Yaskawa INFORM job: t_01_08_23_cylinder_program.JBI

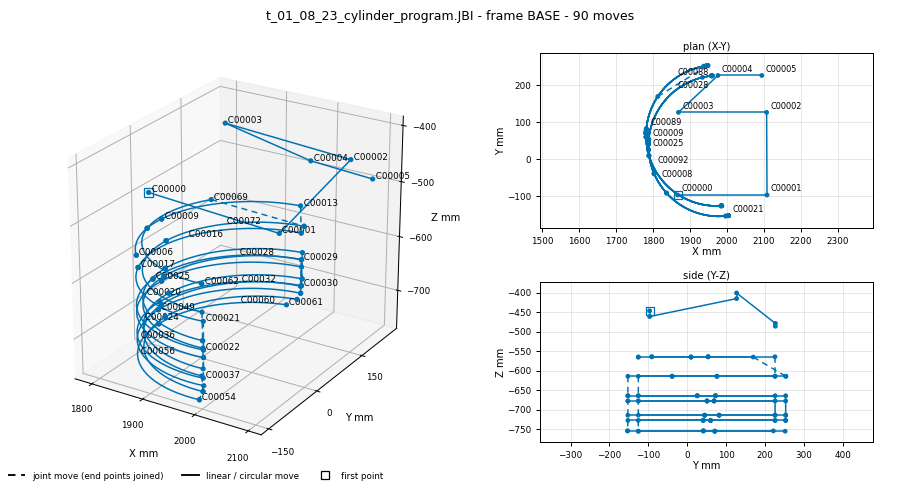
[picture p0: tool path of t_01_08_23_cylinder_program.JBI in frame BASE, 90 of 125 moves have a stored position in this frame; points joined in program order, loops and branches not executed]
/JOB
//NAME t_01_08_23_cylinder_program
//POS
///NPOS 118,0,118,0,0,0
///TOOL 0
///POSTYPE BASE
///RECTAN
///RCONF 0,0,0,0,0,0,0,0,0,0,0,0,0,0,0,0,0,0,0,0,0,0,0,0
C00000=1866.907856,-96.774129,-446.002528,175.000000,-50.248348,92.918411
C00001=2108.409771,-96.774089,-460.785696,175.000000,-50.248348,92.918411
C00002=2107.340894,126.546568,-414.757146,152.980956,5.000000,-5.000000
C00003=1869.210666,126.546528,-400.180371,152.980956,5.000000,-5.000000
C00004=1975.714402,226.206036,-478.423517,175.000000,-60.000000,-90.532197
C00005=2094.376869,226.206056,-485.687257,175.000000,-60.000000,-90.532197
C00006=1836.815666,-91.346481,-564.151000,-138.035050,-90.000000,5.000000
C00007=1836.815666,-91.346481,-564.151000,-138.035050,-90.000000,5.000000
C00008=1813.462641,-59.170193,-564.151000,-150.021884,-90.000000,5.000000
C00009=1788.802698,53.507037,-564.151000,174.711510,-90.000000,5.000000
C00010=1788.802698,53.507037,-564.151000,174.711510,-90.000000,5.000000
C00011=1788.802698,53.507037,-564.151000,174.711510,-90.000000,5.000000
C00012=1799.194788,100.302609,-564.151000,160.247038,-89.999999,5.000000
C00013=1957.618472,225.208793,-564.151000,96.259663,-90.000000,5.000000
C00014=1959.368351,225.392556,-614.195000,95.730143,-89.999999,5.000000
C00015=1959.368351,225.392556,-614.195000,95.730143,-89.999999,5.000000
C00016=1801.888713,107.361045,-614.195000,157.973217,-90.000000,5.000000
C00017=1803.351040,-38.955819,-614.195000,-156.827998,-90.000000,5.000000
C00018=1803.351040,-38.955819,-614.195000,-156.827998,-90.000000,5.000000
C00019=1803.351040,-38.955819,-614.195000,-156.827998,-90.000000,5.000000
C00020=1871.671478,-121.712228,-614.195000,-124.088520,-90.000000,5.000000
C00021=2004.609733,-152.609584,-614.195000,-82.080123,-89.999999,5.000000
C00022=2004.545282,-152.618539,-664.237500,-82.099706,-89.999999,5.000000
C00023=2004.545282,-152.618539,-664.237500,-82.099706,-89.999999,5.000000
C00024=1861.423248,-114.267854,-664.237500,-127.901229,-90.000000,5.000000
C00025=1788.282629,25.448540,-664.237500,-175.000000,-90.000000,5.000000
C00026=1788.282629,25.448540,-664.237500,-175.000000,-90.000000,5.000000
C00027=1788.282629,25.448540,-664.237500,-175.000000,-90.000000,5.000000
C00028=1857.406269,182.970813,-664.237500,129.449763,-90.000000,5.000000
C00029=1960.228639,225.476909,-664.237500,95.470000,-89.999999,5.000000
C00030=1959.424752,225.398207,-714.244000,95.713085,-90.000000,5.000000
C00031=1959.424752,225.398207,-714.244000,95.713085,-90.000000,5.000000
C00032=1860.043911,185.102125,-714.244000,128.429203,-90.000000,5.000000
C00033=1788.186763,44.562490,-714.244000,175.000000,-89.999999,5.000000
C00034=1788.186763,44.562490,-714.244000,175.000000,-89.999999,5.000000
C00035=1788.186763,44.562490,-714.244000,175.000000,-89.999999,5.000000
C00036=1834.273085,-88.461094,-714.244000,-139.192453,-90.000000,5.000000
C00037=2003.923519,-152.703775,-714.244000,-82.288574,-90.000000,5.000000
C00038=2004.586601,-152.612801,-677.657460,-175.000000,-60.000000,97.912848
C00039=2004.586601,-152.612801,-677.657460,-175.000000,-60.000000,97.912848
C00040=1828.234217,-81.102716,-677.657460,175.000000,-60.000000,37.942494
C00041=1788.560641,50.659282,-677.657460,175.000000,-60.000000,-5.000000
C00042=1788.560641,50.659282,-677.657460,175.000000,-60.000000,-5.000000
C00043=1788.560641,50.659282,-677.657460,175.000000,-60.000000,-5.000000
C00044=1853.077163,179.298948,-677.657460,-175.000000,-60.000000,-48.841817
C00045=1960.796933,225.530469,-677.657460,175.000000,-60.000000,-84.701785
C00046=1959.683285,225.423893,-727.621460,175.000000,-60.000000,-84.365103
C00047=1959.683285,225.423893,-727.621460,175.000000,-60.000000,-84.365103
C00048=1855.996123,181.799021,-727.621460,175.000000,-60.000000,-49.998458
C00049=1788.052126,40.732629,-727.621460,-175.000000,-60.000000,-5.000000
C00050=1788.052126,40.732629,-727.621460,-175.000000,-60.000000,-5.000000
C00051=1788.052126,40.732629,-727.621460,-175.000000,-60.000000,-5.000000
C00052=1823.090180,-74.187752,-727.621460,175.000000,-60.000000,35.348569
C00053=2004.520010,-152.622044,-727.621460,175.000000,-60.000000,97.892616
C00054=1996.799177,-153.532136,-754.534960,175.000000,-60.000000,95.552802
C00055=1996.799177,-153.532136,-754.534960,175.000000,-60.000000,95.552802
C00056=1821.172558,-71.433123,-754.534960,175.000000,-60.000000,34.338464
C00057=1788.066435,41.272587,-754.534960,175.000000,-60.000000,-5.000000
C00058=1788.066435,41.272587,-754.534960,175.000000,-60.000000,-5.000000
C00059=1788.066435,41.272587,-754.534960,175.000000,-60.000000,-5.000000
C00060=1858.465261,183.835862,-754.534960,175.000000,-60.000000,-50.961753
C00061=1934.046589,221.110871,-754.534960,175.000000,-60.000000,-76.535293
C00062=1984.729913,-125.856900,-564.850500,-86.117270,-90.000000,5.000000
C00063=1984.729913,-125.856900,-564.850500,-86.117270,-90.000000,5.000000
C00064=1823.365128,-55.081799,-564.850500,-141.247545,-90.000000,5.000000
C00065=1789.445749,9.507244,-564.850500,-163.339420,-90.000000,5.000000
C00066=1789.445749,9.507244,-564.850500,-163.339420,-90.000000,5.000000
C00067=1789.445749,9.507244,-564.850500,-163.339420,-90.000000,5.000000
C00068=1781.565163,70.613527,-564.850500,175.000000,-90.000000,5.000000
C00069=1813.170254,169.308927,-564.850500,146.450271,-90.000000,5.000000
C00070=1948.855670,253.083256,-614.253000,96.933410,-90.000000,5.000000
C00071=1948.855670,253.083256,-614.253000,96.933410,-90.000000,5.000000
C00072=1827.501897,188.241517,-614.253000,139.299547,-89.999999,5.000000
C00073=1781.843312,76.269362,-614.253000,175.000000,-90.000000,5.000000
C00074=1781.843312,76.269362,-614.253000,175.000000,-90.000000,5.000000
C00075=1781.843312,76.269362,-614.253000,175.000000,-90.000000,5.000000
C00076=1839.012225,-72.304280,-614.253000,-134.240439,-89.999999,5.000000
C00077=1984.854502,-125.848403,-614.253000,-86.079688,-89.999999,5.000000
C00078=1985.670166,-125.790746,-664.261500,-85.833603,-90.000000,5.000000
C00079=1985.670166,-125.790746,-664.261500,-85.833603,-90.000000,5.000000
C00080=1817.484848,-47.360560,-664.261500,-144.168682,-89.999999,5.000000
C00081=1781.629678,72.281824,-664.261500,175.000000,-90.000000,5.000000
C00082=1781.629678,72.281824,-664.261500,175.000000,-90.000000,5.000000
C00083=1781.629678,72.281824,-664.261500,175.000000,-90.000000,5.000000
C00084=1848.588115,209.196904,-664.261500,130.343854,-90.000000,5.000000
C00085=1946.287238,252.753181,-664.261500,97.712735,-90.000000,5.000000
C00086=1946.337263,252.759949,-714.232500,97.697544,-89.999999,5.000000
C00087=1946.337263,252.759949,-714.232500,97.697544,-89.999999,5.000000
C00088=1857.182730,216.079242,-714.232500,127.029772,-90.000000,5.000000
C00089=1782.269209,81.696835,-714.232500,174.693933,-89.999999,5.000000
C00090=1782.269209,81.696835,-714.232500,174.693933,-89.999999,5.000000
C00091=1782.269209,81.696835,-714.232500,174.693933,-89.999999,5.000000
C00092=1801.115148,-20.170739,-714.232500,-153.731021,-90.000000,5.000000
C00093=1986.144740,-125.755579,-714.232500,-85.690389,-89.999999,5.000000
C00094=1986.131450,-125.756580,-677.631960,175.000000,-60.000000,94.305599
C00095=1986.131450,-125.756580,-677.631960,175.000000,-60.000000,94.305599
C00096=1813.820766,-42.101735,-677.631960,-175.000000,-60.000000,33.902326
C00097=1781.507638,68.635230,-677.631960,175.000000,-60.000000,-5.000000
C00098=1781.507638,68.635230,-677.631960,175.000000,-60.000000,-5.000000
C00099=1781.507638,68.635230,-677.631960,175.000000,-60.000000,-5.000000
C00100=1843.052224,204.306842,-677.631960,175.000000,-60.000000,-47.433091
C00101=1945.255131,252.610524,-677.631960,175.000000,-60.000000,-81.973701
C00102=1945.341344,252.622661,-727.629960,175.000000,-60.000000,-81.999903
C00103=1945.341344,252.622661,-727.629960,175.000000,-60.000000,-81.999903
C00104=1840.373702,201.798651,-727.629960,175.000000,-60.000000,-46.328736
C00105=1781.500906,59.837692,-727.629960,175.000000,-60.000000,5.000000
C00106=1781.500906,59.837692,-727.629960,175.000000,-60.000000,5.000000
C00107=1781.500906,59.837692,-727.629960,175.000000,-60.000000,5.000000
C00108=1812.240335,-39.711348,-727.629960,175.000000,-60.000000,33.039921
C00109=1983.737597,-125.921646,-727.629960,175.000000,-60.000000,93.583460
C00110=1985.619988,-125.794394,-755.330960,175.000000,-60.000000,94.151256
C00111=1985.619988,-125.794394,-755.330960,175.000000,-60.000000,94.151256
C00112=1814.137027,-42.570833,-755.330960,175.000000,-60.000000,34.072588
C00113=1781.563747,70.572080,-755.330960,175.000000,-60.000000,-5.000000
C00114=1781.563747,70.572080,-755.330960,175.000000,-60.000000,-5.000000
C00115=1781.563747,70.572080,-755.330960,175.000000,-60.000000,-5.000000
C00116=1897.879181,239.522892,-755.330960,175.000000,-60.000000,-67.140613
C00117=1937.434389,251.341235,-755.330960,175.000000,-60.000000,-79.589100
///POSTYPE PULSE
///PULSE
EX00000=98304.0
EX00001=99328.0
EX00002=282624.0
///POSTYPE PULSE
///PULSE
EC00000=98304.0
EC00001=98304.0
EC00002=98304.0
EC00003=98304.0
EC00004=98304.0
EC00005=98304.0
EC00006=99328.0
EC00007=99328.0
EC00008=99328.0
EC00009=99328.0
EC00010=99328.0
EC00011=99328.0
EC00012=99328.0
EC00013=99328.0
EC00014=99328.0
EC00015=99328.0
EC00016=99328.0
EC00017=99328.0
EC00018=99328.0
EC00019=99328.0
EC00020=99328.0
EC00021=99328.0
EC00022=99328.0
EC00023=99328.0
EC00024=99328.0
EC00025=99328.0
EC00026=99328.0
EC00027=99328.0
EC00028=99328.0
EC00029=99328.0
EC00030=99328.0
EC00031=99328.0
EC00032=99328.0
EC00033=99328.0
EC00034=99328.0
EC00035=99328.0
EC00036=99328.0
EC00037=99328.0
EC00038=99328.0
EC00039=99328.0
EC00040=99328.0
EC00041=99328.0
EC00042=99328.0
EC00043=99328.0
EC00044=99328.0
EC00045=99328.0
EC00046=99328.0
EC00047=99328.0
EC00048=99328.0
EC00049=99328.0
EC00050=99328.0
EC00051=99328.0
EC00052=99328.0
EC00053=99328.0
EC00054=99328.0
EC00055=99328.0
EC00056=99328.0
EC00057=99328.0
EC00058=99328.0
EC00059=99328.0
EC00060=99328.0
EC00061=99328.0
EC00062=282624.0
EC00063=282624.0
EC00064=282624.0
EC00065=282624.0
EC00066=282624.0
EC00067=282624.0
EC00068=282624.0
EC00069=282624.0
EC00070=282624.0
EC00071=282624.0
EC00072=282624.0
EC00073=282624.0
EC00074=282624.0
EC00075=282624.0
EC00076=282624.0
EC00077=282624.0
EC00078=282624.0
EC00079=282624.0
EC00080=282624.0
EC00081=282624.0
EC00082=282624.0
EC00083=282624.0
EC00084=282624.0
EC00085=282624.0
EC00086=282624.0
EC00087=282624.0
EC00088=282624.0
EC00089=282624.0
EC00090=282624.0
EC00091=282624.0
EC00092=282624.0
EC00093=282624.0
EC00094=282624.0
EC00095=282624.0
EC00096=282624.0
EC00097=282624.0
EC00098=282624.0
EC00099=282624.0
EC00100=282624.0
EC00101=282624.0
EC00102=282624.0
EC00103=282624.0
EC00104=282624.0
EC00105=282624.0
EC00106=282624.0
EC00107=282624.0
EC00108=282624.0
EC00109=282624.0
EC00110=282624.0
EC00111=282624.0
EC00112=282624.0
EC00113=282624.0
EC00114=282624.0
EC00115=282624.0
EC00116=282624.0
EC00117=282624.0
//INST
///DATE 2023/08/16 12:22
///ATTR SC,RW,RJ
////FRAME BASE
///GROUP1 RB1,ST1
NOP
MOVJ P009 EX000 VJ=15.00
MOVJ C00000 EC00000 VJ=15.0
CALL JOB:SPYON
MOVL C00001 EC00001 V=150.0
MOVL C00002 EC00002 V=150.0
MOVL C00003 EC00003 V=150.0
MOVL C00004 EC00004 V=150.0
MOVL C00005 EC00005 V=150.0
CALL JOB:SPYOF
MOVJ P009 VJ=15.00
MOVL P009 EX00000 V=150.0
MOVJ C00006 EC00006 VJ=15.0
CALL JOB:SPYON
MOVC C00007 EC00007 V=150.0
MOVC C00008 EC00008 V=150.0
MOVC C00009 EC00009 V=150.0
MOVJ C00010 EC00010 VJ=15.0
MOVC C00011 EC00011 V=150.0
MOVC C00012 EC00012 V=150.0
MOVC C00013 EC00013 V=150.0
MOVJ C00014 EC00014 VJ=15.0
MOVC C00015 EC00015 V=150.0
MOVC C00016 EC00016 V=150.0
MOVC C00017 EC00017 V=150.0
MOVJ C00018 EC00018 VJ=15.0
MOVC C00019 EC00019 V=150.0
MOVC C00020 EC00020 V=150.0
MOVC C00021 EC00021 V=150.0
MOVJ C00022 EC00022 VJ=15.0
MOVC C00023 EC00023 V=150.0
MOVC C00024 EC00024 V=150.0
MOVC C00025 EC00025 V=150.0
MOVJ C00026 EC00026 VJ=15.0
MOVC C00027 EC00027 V=150.0
MOVC C00028 EC00028 V=150.0
MOVC C00029 EC00029 V=150.0
MOVJ C00030 EC00030 VJ=15.0
MOVC C00031 EC00031 V=150.0
MOVC C00032 EC00032 V=150.0
MOVC C00033 EC00033 V=150.0
MOVJ C00034 EC00034 VJ=15.0
MOVC C00035 EC00035 V=150.0
MOVC C00036 EC00036 V=150.0
MOVC C00037 EC00037 V=150.0
MOVJ C00038 EC00038 VJ=15.0
MOVC C00039 EC00039 V=150.0
MOVC C00040 EC00040 V=150.0
MOVC C00041 EC00041 V=150.0
MOVJ C00042 EC00042 VJ=15.0
MOVC C00043 EC00043 V=150.0
MOVC C00044 EC00044 V=150.0
MOVC C00045 EC00045 V=150.0
MOVJ C00046 EC00046 VJ=15.0
MOVC C00047 EC00047 V=150.0
MOVC C00048 EC00048 V=150.0
MOVC C00049 EC00049 V=150.0
MOVJ C00050 EC00050 VJ=15.0
MOVC C00051 EC00051 V=150.0
MOVC C00052 EC00052 V=150.0
MOVC C00053 EC00053 V=150.0
MOVJ C00054 EC00054 VJ=15.0
MOVC C00055 EC00055 V=150.0
MOVC C00056 EC00056 V=150.0
MOVC C00057 EC00057 V=150.0
MOVJ C00058 EC00058 VJ=15.0
MOVC C00059 EC00059 V=150.0
MOVC C00060 EC00060 V=150.0
MOVC C00061 EC00061 V=150.0
CALL JOB:SPYOF
MOVJ P009 VJ=15.00
MOVL P009 EX00001 V=150.0
MOVJ C00062 EC00062 VJ=15.0
CALL JOB:SPYON
MOVC C00063 EC00063 V=150.0
MOVC C00064 EC00064 V=150.0
MOVC C00065 EC00065 V=150.0
MOVJ C00066 EC00066 VJ=15.0
MOVC C00067 EC00067 V=150.0
MOVC C00068 EC00068 V=150.0
MOVC C00069 EC00069 V=150.0
MOVJ C00070 EC00070 VJ=15.0
MOVC C00071 EC00071 V=150.0
MOVC C00072 EC00072 V=150.0
MOVC C00073 EC00073 V=150.0
MOVJ C00074 EC00074 VJ=15.0
MOVC C00075 EC00075 V=150.0
MOVC C00076 EC00076 V=150.0
MOVC C00077 EC00077 V=150.0
MOVJ C00078 EC00078 VJ=15.0
MOVC C00079 EC00079 V=150.0
MOVC C00080 EC00080 V=150.0
MOVC C00081 EC00081 V=150.0
MOVJ C00082 EC00082 VJ=15.0
MOVC C00083 EC00083 V=150.0
MOVC C00084 EC00084 V=150.0
MOVC C00085 EC00085 V=150.0
MOVJ C00086 EC00086 VJ=15.0
MOVC C00087 EC00087 V=150.0
MOVC C00088 EC00088 V=150.0
MOVC C00089 EC00089 V=150.0
MOVJ C00090 EC00090 VJ=15.0
MOVC C00091 EC00091 V=150.0
MOVC C00092 EC00092 V=150.0
MOVC C00093 EC00093 V=150.0
MOVJ C00094 EC00094 VJ=15.0
MOVC C00095 EC00095 V=150.0
MOVC C00096 EC00096 V=150.0
MOVC C00097 EC00097 V=150.0
MOVJ C00098 EC00098 VJ=15.0
MOVC C00099 EC00099 V=150.0
MOVC C00100 EC00100 V=150.0
MOVC C00101 EC00101 V=150.0
MOVJ C00102 EC00102 VJ=15.0
MOVC C00103 EC00103 V=150.0
MOVC C00104 EC00104 V=150.0
MOVC C00105 EC00105 V=150.0
MOVJ C00106 EC00106 VJ=15.0
MOVC C00107 EC00107 V=150.0
MOVC C00108 EC00108 V=150.0
MOVC C00109 EC00109 V=150.0
MOVJ C00110 EC00110 VJ=15.0
MOVC C00111 EC00111 V=150.0
MOVC C00112 EC00112 V=150.0
MOVC C00113 EC00113 V=150.0
MOVJ C00114 EC00114 VJ=15.0
MOVC C00115 EC00115 V=150.0
MOVC C00116 EC00116 V=150.0
MOVC C00117 EC00117 V=150.0
CALL JOB:SPYOF
MOVJ P009 VJ=15.00
MOVL P009 EX00002 V=150.0
END
